(* Visualisation SCHO2_GR4
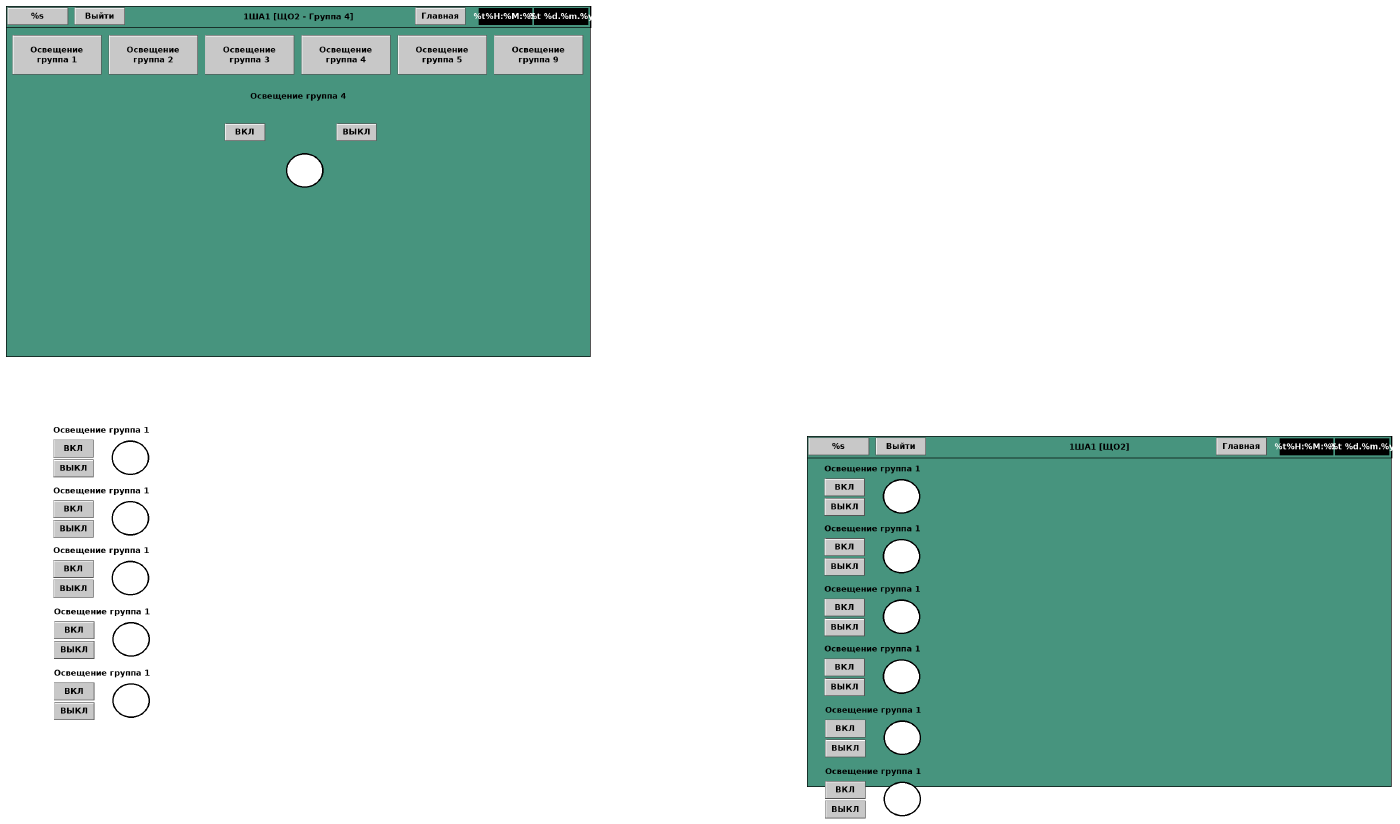
rectangle at (0,0)-(802,30): text "1ША1 [ЩО2 - Группа 4]"
button at (2,2)-(85,26): text "%s"; shows VHOD.User
button at (94,2)-(163,26): text "Выйти"; toggles VHOD.bVihod; opens A0_START_WINDOW
button at (561,2)-(630,26): text "Главная"; opens A1_START_WINDOW
rectangle at (648,3)-(721,26): text "%t%H:%M:%S"
rectangle at (724,3)-(798,26): text "%t %d.%m.%y"
rectangle at (6,107)-(796,141): text "Освещение группа 4"
button at (300,161)-(355,185): text "ВКЛ"; toggles .bK152_1SHA1_SCHO2_LIGHT_GR4_ON
button at (453,161)-(508,185): text "ВЫКЛ"; taps .bK152_1SHA1_SCHO2_LIGHT_GR4_OFF
ellipse at (384,202)-(435,249): alarm colour if .K152_1SHA1_SCHO2_KM_GR4
rectangle at (45,570)-(217,594): text "Освещение группа 1"
button at (65,595)-(120,619): text "ВКЛ"; toggles .bK152_1SHA1_SCHAO1_LIGHT_GR5_ON
button at (65,622)-(120,646): text "ВЫКЛ"; taps .bK152_1SHA1_SCHAO1_LIGHT_GR5_OFF
ellipse at (145,596)-(196,643): alarm colour if .K152_1SHA1_SCHAO1_LIGHT_GR5
rectangle at (45,653)-(217,677): text "Освещение группа 1"
button at (65,678)-(120,702): text "ВКЛ"; toggles .bK152_1SHA1_SCHAO1_LIGHT_GR5_ON
button at (65,705)-(120,729): text "ВЫКЛ"; taps .bK152_1SHA1_SCHAO1_LIGHT_GR5_OFF
ellipse at (145,679)-(196,726): alarm colour if .K152_1SHA1_SCHAO1_LIGHT_GR5
rectangle at (45,735)-(217,759): text "Освещение группа 1"
button at (65,760)-(120,784): text "ВКЛ"; toggles .bK152_1SHA1_SCHAO1_LIGHT_GR5_ON
button at (65,787)-(120,811): text "ВЫКЛ"; taps .bK152_1SHA1_SCHAO1_LIGHT_GR5_OFF
ellipse at (145,761)-(196,808): alarm colour if .K152_1SHA1_SCHAO1_LIGHT_GR5
rectangle at (46,819)-(218,843): text "Освещение группа 1"
button at (66,844)-(121,868): text "ВКЛ"; toggles .bK152_1SHA1_SCHAO1_LIGHT_GR5_ON
button at (66,871)-(121,895): text "ВЫКЛ"; taps .bK152_1SHA1_SCHAO1_LIGHT_GR5_OFF
ellipse at (146,845)-(197,892): alarm colour if .K152_1SHA1_SCHAO1_LIGHT_GR5
rectangle at (46,903)-(218,927): text "Освещение группа 1"
button at (66,928)-(121,952): text "ВКЛ"; toggles .bK152_1SHA1_SCHAO1_LIGHT_GR5_ON
button at (66,955)-(121,979): text "ВЫКЛ"; taps .bK152_1SHA1_SCHAO1_LIGHT_GR5_OFF
ellipse at (146,929)-(197,976): alarm colour if .K152_1SHA1_SCHAO1_LIGHT_GR5
rectangle at (1098,590)-(1900,620): text "1ША1 [ЩО2]"
button at (1100,592)-(1183,616): text "%s"; shows VHOD.User
button at (1192,592)-(1261,616): text "Выйти"; toggles VHOD.bVihod; opens A0_START_WINDOW
button at (1659,592)-(1728,616): text "Главная"; opens A1_START_WINDOW
rectangle at (1746,593)-(1819,616): text "%t%H:%M:%S"
rectangle at (1822,593)-(1896,616): text "%t %d.%m.%y"
rectangle at (1102,623)-(1274,647): text "Освещение группа 1"
button at (1122,648)-(1177,672): text "ВКЛ"; toggles .bK152_1SHA1_SCHAO1_LIGHT_GR5_ON
button at (1122,675)-(1177,699): text "ВЫКЛ"; taps .bK152_1SHA1_SCHAO1_LIGHT_GR5_OFF
ellipse at (1202,649)-(1253,696): alarm colour if .K152_1SHA1_SCHAO1_LIGHT_GR5
rectangle at (1102,705)-(1274,729): text "Освещение группа 1"
button at (1122,730)-(1177,754): text "ВКЛ"; toggles .bK152_1SHA1_SCHAO1_LIGHT_GR5_ON
button at (1122,757)-(1177,781): text "ВЫКЛ"; taps .bK152_1SHA1_SCHAO1_LIGHT_GR5_OFF
ellipse at (1202,731)-(1253,778): alarm colour if .K152_1SHA1_SCHAO1_LIGHT_GR5
rectangle at (1102,788)-(1274,812): text "Освещение группа 1"
button at (1122,813)-(1177,837): text "ВКЛ"; toggles .bK152_1SHA1_SCHAO1_LIGHT_GR5_ON
button at (1122,840)-(1177,864): text "ВЫКЛ"; taps .bK152_1SHA1_SCHAO1_LIGHT_GR5_OFF
ellipse at (1202,814)-(1253,861): alarm colour if .K152_1SHA1_SCHAO1_LIGHT_GR5
rectangle at (1102,870)-(1274,894): text "Освещение группа 1"
button at (1122,895)-(1177,919): text "ВКЛ"; toggles .bK152_1SHA1_SCHAO1_LIGHT_GR5_ON
button at (1122,922)-(1177,946): text "ВЫКЛ"; taps .bK152_1SHA1_SCHAO1_LIGHT_GR5_OFF
ellipse at (1202,896)-(1253,943): alarm colour if .K152_1SHA1_SCHAO1_LIGHT_GR5
rectangle at (1103,954)-(1275,978): text "Освещение группа 1"
button at (1123,979)-(1178,1003): text "ВКЛ"; toggles .bK152_1SHA1_SCHAO1_LIGHT_GR5_ON
button at (1123,1006)-(1178,1030): text "ВЫКЛ"; taps .bK152_1SHA1_SCHAO1_LIGHT_GR5_OFF
ellipse at (1203,980)-(1254,1027): alarm colour if .K152_1SHA1_SCHAO1_LIGHT_GR5
rectangle at (1103,1038)-(1275,1062): text "Освещение группа 1"
button at (1123,1063)-(1178,1087): text "ВКЛ"; toggles .bK152_1SHA1_SCHAO1_LIGHT_GR5_ON
button at (1123,1090)-(1178,1114): text "ВЫКЛ"; taps .bK152_1SHA1_SCHAO1_LIGHT_GR5_OFF
ellipse at (1203,1064)-(1254,1111): alarm colour if .K152_1SHA1_SCHAO1_LIGHT_GR5
button at (9,40)-(131,94): text "Освещение / группа 1"; opens SCHO2_GR1
button at (141,40)-(263,94): text "Освещение / группа 2"; opens SCHO2_GR2
button at (273,40)-(395,94): text "Освещение / группа 3"; opens SCHO2_GR3
button at (405,40)-(527,94): text "Освещение / группа 4"; opens SCHO2_GR4
button at (537,40)-(659,94): text "Освещение / группа 5"; opens SCHO2_GR5
button at (669,40)-(791,94): text "Освещение / группа 9"; opens SCHO2_GR9
2 more shapes without text or variables
14 elements of other kinds (tables, trends, ...) not read
*)

(* Visualisation SCHO2_GR5
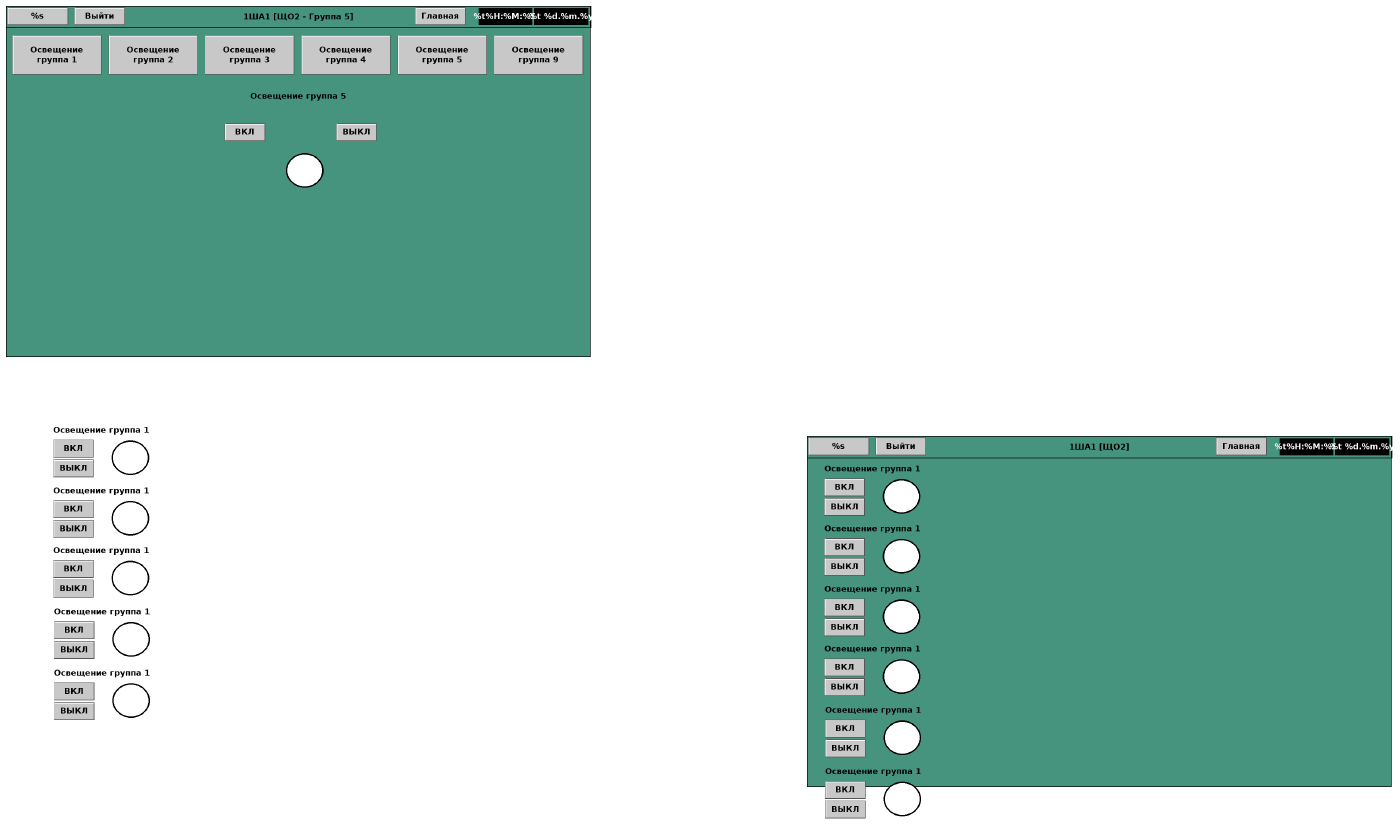
rectangle at (0,0)-(802,30): text "1ША1 [ЩО2 - Группа 5]"
button at (2,2)-(85,26): text "%s"; shows VHOD.User
button at (94,2)-(163,26): text "Выйти"; toggles VHOD.bVihod; opens A0_START_WINDOW
button at (561,2)-(630,26): text "Главная"; opens A1_START_WINDOW
rectangle at (648,3)-(721,26): text "%t%H:%M:%S"
rectangle at (724,3)-(798,26): text "%t %d.%m.%y"
rectangle at (6,107)-(796,141): text "Освещение группа 5"
button at (300,161)-(355,185): text "ВКЛ"; toggles .bK152_1SHA1_SCHO2_LIGHT_GR5_ON
button at (453,161)-(508,185): text "ВЫКЛ"; taps .bK152_1SHA1_SCHO2_LIGHT_GR5_OFF
ellipse at (384,202)-(435,249): alarm colour if .K152_1SHA1_SCHO2_KM_GR5
rectangle at (45,570)-(217,594): text "Освещение группа 1"
button at (65,595)-(120,619): text "ВКЛ"; toggles .bK152_1SHA1_SCHAO1_LIGHT_GR5_ON
button at (65,622)-(120,646): text "ВЫКЛ"; taps .bK152_1SHA1_SCHAO1_LIGHT_GR5_OFF
ellipse at (145,596)-(196,643): alarm colour if .K152_1SHA1_SCHAO1_LIGHT_GR5
rectangle at (45,653)-(217,677): text "Освещение группа 1"
button at (65,678)-(120,702): text "ВКЛ"; toggles .bK152_1SHA1_SCHAO1_LIGHT_GR5_ON
button at (65,705)-(120,729): text "ВЫКЛ"; taps .bK152_1SHA1_SCHAO1_LIGHT_GR5_OFF
ellipse at (145,679)-(196,726): alarm colour if .K152_1SHA1_SCHAO1_LIGHT_GR5
rectangle at (45,735)-(217,759): text "Освещение группа 1"
button at (65,760)-(120,784): text "ВКЛ"; toggles .bK152_1SHA1_SCHAO1_LIGHT_GR5_ON
button at (65,787)-(120,811): text "ВЫКЛ"; taps .bK152_1SHA1_SCHAO1_LIGHT_GR5_OFF
ellipse at (145,761)-(196,808): alarm colour if .K152_1SHA1_SCHAO1_LIGHT_GR5
rectangle at (46,819)-(218,843): text "Освещение группа 1"
button at (66,844)-(121,868): text "ВКЛ"; toggles .bK152_1SHA1_SCHAO1_LIGHT_GR5_ON
button at (66,871)-(121,895): text "ВЫКЛ"; taps .bK152_1SHA1_SCHAO1_LIGHT_GR5_OFF
ellipse at (146,845)-(197,892): alarm colour if .K152_1SHA1_SCHAO1_LIGHT_GR5
rectangle at (46,903)-(218,927): text "Освещение группа 1"
button at (66,928)-(121,952): text "ВКЛ"; toggles .bK152_1SHA1_SCHAO1_LIGHT_GR5_ON
button at (66,955)-(121,979): text "ВЫКЛ"; taps .bK152_1SHA1_SCHAO1_LIGHT_GR5_OFF
ellipse at (146,929)-(197,976): alarm colour if .K152_1SHA1_SCHAO1_LIGHT_GR5
rectangle at (1098,590)-(1900,620): text "1ША1 [ЩО2]"
button at (1100,592)-(1183,616): text "%s"; shows VHOD.User
button at (1192,592)-(1261,616): text "Выйти"; toggles VHOD.bVihod; opens A0_START_WINDOW
button at (1659,592)-(1728,616): text "Главная"; opens A1_START_WINDOW
rectangle at (1746,593)-(1819,616): text "%t%H:%M:%S"
rectangle at (1822,593)-(1896,616): text "%t %d.%m.%y"
rectangle at (1102,623)-(1274,647): text "Освещение группа 1"
button at (1122,648)-(1177,672): text "ВКЛ"; toggles .bK152_1SHA1_SCHAO1_LIGHT_GR5_ON
button at (1122,675)-(1177,699): text "ВЫКЛ"; taps .bK152_1SHA1_SCHAO1_LIGHT_GR5_OFF
ellipse at (1202,649)-(1253,696): alarm colour if .K152_1SHA1_SCHAO1_LIGHT_GR5
rectangle at (1102,705)-(1274,729): text "Освещение группа 1"
button at (1122,730)-(1177,754): text "ВКЛ"; toggles .bK152_1SHA1_SCHAO1_LIGHT_GR5_ON
button at (1122,757)-(1177,781): text "ВЫКЛ"; taps .bK152_1SHA1_SCHAO1_LIGHT_GR5_OFF
ellipse at (1202,731)-(1253,778): alarm colour if .K152_1SHA1_SCHAO1_LIGHT_GR5
rectangle at (1102,788)-(1274,812): text "Освещение группа 1"
button at (1122,813)-(1177,837): text "ВКЛ"; toggles .bK152_1SHA1_SCHAO1_LIGHT_GR5_ON
button at (1122,840)-(1177,864): text "ВЫКЛ"; taps .bK152_1SHA1_SCHAO1_LIGHT_GR5_OFF
ellipse at (1202,814)-(1253,861): alarm colour if .K152_1SHA1_SCHAO1_LIGHT_GR5
rectangle at (1102,870)-(1274,894): text "Освещение группа 1"
button at (1122,895)-(1177,919): text "ВКЛ"; toggles .bK152_1SHA1_SCHAO1_LIGHT_GR5_ON
button at (1122,922)-(1177,946): text "ВЫКЛ"; taps .bK152_1SHA1_SCHAO1_LIGHT_GR5_OFF
ellipse at (1202,896)-(1253,943): alarm colour if .K152_1SHA1_SCHAO1_LIGHT_GR5
rectangle at (1103,954)-(1275,978): text "Освещение группа 1"
button at (1123,979)-(1178,1003): text "ВКЛ"; toggles .bK152_1SHA1_SCHAO1_LIGHT_GR5_ON
button at (1123,1006)-(1178,1030): text "ВЫКЛ"; taps .bK152_1SHA1_SCHAO1_LIGHT_GR5_OFF
ellipse at (1203,980)-(1254,1027): alarm colour if .K152_1SHA1_SCHAO1_LIGHT_GR5
rectangle at (1103,1038)-(1275,1062): text "Освещение группа 1"
button at (1123,1063)-(1178,1087): text "ВКЛ"; toggles .bK152_1SHA1_SCHAO1_LIGHT_GR5_ON
button at (1123,1090)-(1178,1114): text "ВЫКЛ"; taps .bK152_1SHA1_SCHAO1_LIGHT_GR5_OFF
ellipse at (1203,1064)-(1254,1111): alarm colour if .K152_1SHA1_SCHAO1_LIGHT_GR5
button at (9,40)-(131,94): text "Освещение / группа 1"; opens SCHO2_GR1
button at (141,40)-(263,94): text "Освещение / группа 2"; opens SCHO2_GR2
button at (273,40)-(395,94): text "Освещение / группа 3"; opens SCHO2_GR3
button at (405,40)-(527,94): text "Освещение / группа 4"; opens SCHO2_GR4
button at (537,40)-(659,94): text "Освещение / группа 5"; opens SCHO2_GR5
button at (669,40)-(791,94): text "Освещение / группа 9"; opens SCHO2_GR9
2 more shapes without text or variables
14 elements of other kinds (tables, trends, ...) not read
*)

(* Visualisation SCHO2_GR9
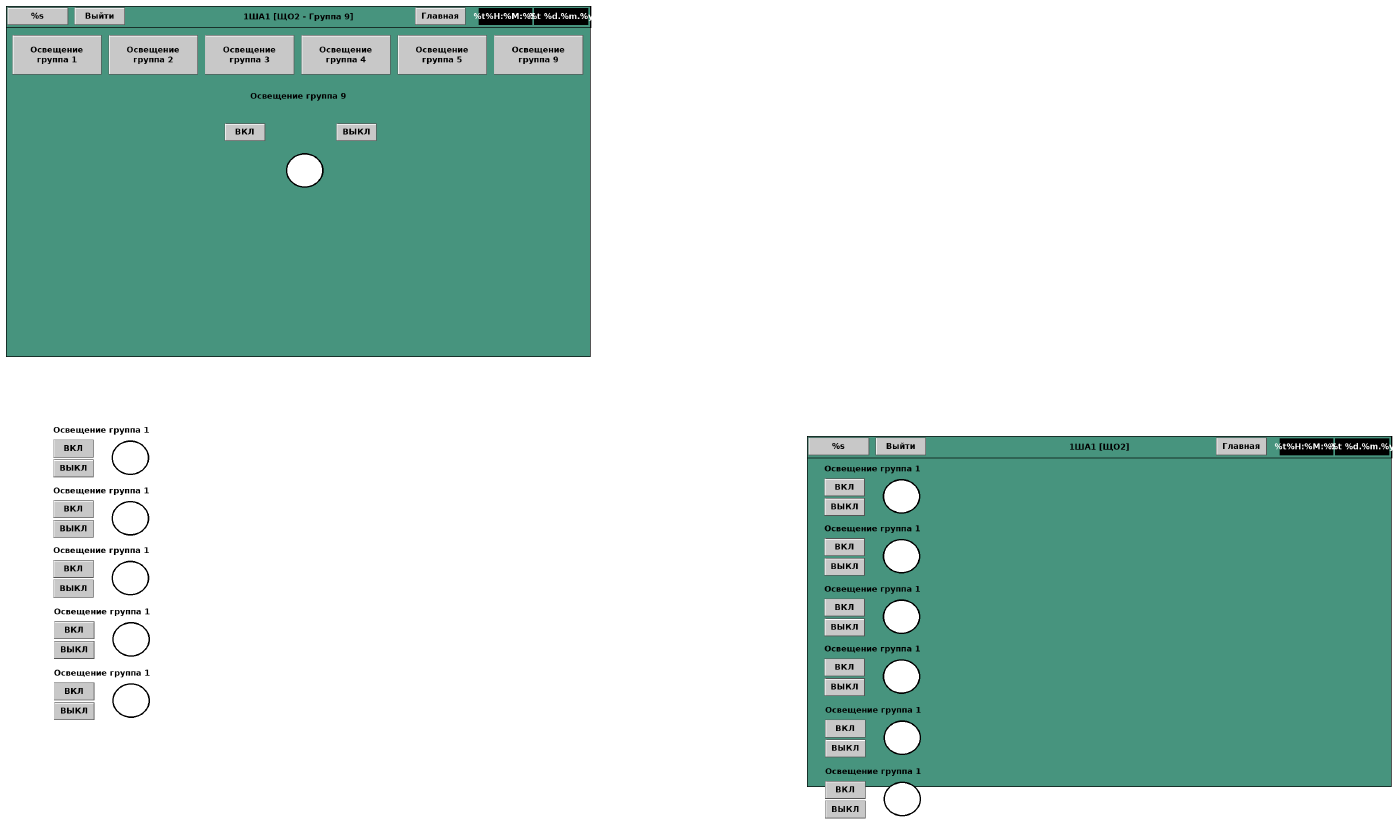
rectangle at (0,0)-(802,30): text "1ША1 [ЩО2 - Группа 9]"
button at (2,2)-(85,26): text "%s"; shows VHOD.User
button at (94,2)-(163,26): text "Выйти"; toggles VHOD.bVihod; opens A0_START_WINDOW
button at (561,2)-(630,26): text "Главная"; opens A1_START_WINDOW
rectangle at (648,3)-(721,26): text "%t%H:%M:%S"
rectangle at (724,3)-(798,26): text "%t %d.%m.%y"
rectangle at (6,107)-(796,141): text "Освещение группа 9"
button at (300,161)-(355,185): text "ВКЛ"; toggles .bK152_1SHA1_SCHO2_LIGHT_GR9_ON
button at (453,161)-(508,185): text "ВЫКЛ"; taps .bK152_1SHA1_SCHO2_LIGHT_GR9_OFF
ellipse at (384,202)-(435,249): alarm colour if .K152_1SHA1_SCHO2_KM_GR9
rectangle at (45,570)-(217,594): text "Освещение группа 1"
button at (65,595)-(120,619): text "ВКЛ"; toggles .bK152_1SHA1_SCHAO1_LIGHT_GR5_ON
button at (65,622)-(120,646): text "ВЫКЛ"; taps .bK152_1SHA1_SCHAO1_LIGHT_GR5_OFF
ellipse at (145,596)-(196,643): alarm colour if .K152_1SHA1_SCHAO1_LIGHT_GR5
rectangle at (45,653)-(217,677): text "Освещение группа 1"
button at (65,678)-(120,702): text "ВКЛ"; toggles .bK152_1SHA1_SCHAO1_LIGHT_GR5_ON
button at (65,705)-(120,729): text "ВЫКЛ"; taps .bK152_1SHA1_SCHAO1_LIGHT_GR5_OFF
ellipse at (145,679)-(196,726): alarm colour if .K152_1SHA1_SCHAO1_LIGHT_GR5
rectangle at (45,735)-(217,759): text "Освещение группа 1"
button at (65,760)-(120,784): text "ВКЛ"; toggles .bK152_1SHA1_SCHAO1_LIGHT_GR5_ON
button at (65,787)-(120,811): text "ВЫКЛ"; taps .bK152_1SHA1_SCHAO1_LIGHT_GR5_OFF
ellipse at (145,761)-(196,808): alarm colour if .K152_1SHA1_SCHAO1_LIGHT_GR5
rectangle at (46,819)-(218,843): text "Освещение группа 1"
button at (66,844)-(121,868): text "ВКЛ"; toggles .bK152_1SHA1_SCHAO1_LIGHT_GR5_ON
button at (66,871)-(121,895): text "ВЫКЛ"; taps .bK152_1SHA1_SCHAO1_LIGHT_GR5_OFF
ellipse at (146,845)-(197,892): alarm colour if .K152_1SHA1_SCHAO1_LIGHT_GR5
rectangle at (46,903)-(218,927): text "Освещение группа 1"
button at (66,928)-(121,952): text "ВКЛ"; toggles .bK152_1SHA1_SCHAO1_LIGHT_GR5_ON
button at (66,955)-(121,979): text "ВЫКЛ"; taps .bK152_1SHA1_SCHAO1_LIGHT_GR5_OFF
ellipse at (146,929)-(197,976): alarm colour if .K152_1SHA1_SCHAO1_LIGHT_GR5
rectangle at (1098,590)-(1900,620): text "1ША1 [ЩО2]"
button at (1100,592)-(1183,616): text "%s"; shows VHOD.User
button at (1192,592)-(1261,616): text "Выйти"; toggles VHOD.bVihod; opens A0_START_WINDOW
button at (1659,592)-(1728,616): text "Главная"; opens A1_START_WINDOW
rectangle at (1746,593)-(1819,616): text "%t%H:%M:%S"
rectangle at (1822,593)-(1896,616): text "%t %d.%m.%y"
rectangle at (1102,623)-(1274,647): text "Освещение группа 1"
button at (1122,648)-(1177,672): text "ВКЛ"; toggles .bK152_1SHA1_SCHAO1_LIGHT_GR5_ON
button at (1122,675)-(1177,699): text "ВЫКЛ"; taps .bK152_1SHA1_SCHAO1_LIGHT_GR5_OFF
ellipse at (1202,649)-(1253,696): alarm colour if .K152_1SHA1_SCHAO1_LIGHT_GR5
rectangle at (1102,705)-(1274,729): text "Освещение группа 1"
button at (1122,730)-(1177,754): text "ВКЛ"; toggles .bK152_1SHA1_SCHAO1_LIGHT_GR5_ON
button at (1122,757)-(1177,781): text "ВЫКЛ"; taps .bK152_1SHA1_SCHAO1_LIGHT_GR5_OFF
ellipse at (1202,731)-(1253,778): alarm colour if .K152_1SHA1_SCHAO1_LIGHT_GR5
rectangle at (1102,788)-(1274,812): text "Освещение группа 1"
button at (1122,813)-(1177,837): text "ВКЛ"; toggles .bK152_1SHA1_SCHAO1_LIGHT_GR5_ON
button at (1122,840)-(1177,864): text "ВЫКЛ"; taps .bK152_1SHA1_SCHAO1_LIGHT_GR5_OFF
ellipse at (1202,814)-(1253,861): alarm colour if .K152_1SHA1_SCHAO1_LIGHT_GR5
rectangle at (1102,870)-(1274,894): text "Освещение группа 1"
button at (1122,895)-(1177,919): text "ВКЛ"; toggles .bK152_1SHA1_SCHAO1_LIGHT_GR5_ON
button at (1122,922)-(1177,946): text "ВЫКЛ"; taps .bK152_1SHA1_SCHAO1_LIGHT_GR5_OFF
ellipse at (1202,896)-(1253,943): alarm colour if .K152_1SHA1_SCHAO1_LIGHT_GR5
rectangle at (1103,954)-(1275,978): text "Освещение группа 1"
button at (1123,979)-(1178,1003): text "ВКЛ"; toggles .bK152_1SHA1_SCHAO1_LIGHT_GR5_ON
button at (1123,1006)-(1178,1030): text "ВЫКЛ"; taps .bK152_1SHA1_SCHAO1_LIGHT_GR5_OFF
ellipse at (1203,980)-(1254,1027): alarm colour if .K152_1SHA1_SCHAO1_LIGHT_GR5
rectangle at (1103,1038)-(1275,1062): text "Освещение группа 1"
button at (1123,1063)-(1178,1087): text "ВКЛ"; toggles .bK152_1SHA1_SCHAO1_LIGHT_GR5_ON
button at (1123,1090)-(1178,1114): text "ВЫКЛ"; taps .bK152_1SHA1_SCHAO1_LIGHT_GR5_OFF
ellipse at (1203,1064)-(1254,1111): alarm colour if .K152_1SHA1_SCHAO1_LIGHT_GR5
button at (9,40)-(131,94): text "Освещение / группа 1"; opens SCHO2_GR1
button at (141,40)-(263,94): text "Освещение / группа 2"; opens SCHO2_GR2
button at (273,40)-(395,94): text "Освещение / группа 3"; opens SCHO2_GR3
button at (405,40)-(527,94): text "Освещение / группа 4"; opens SCHO2_GR4
button at (537,40)-(659,94): text "Освещение / группа 5"; opens SCHO2_GR5
button at (669,40)-(791,94): text "Освещение / группа 9"; opens SCHO2_GR9
2 more shapes without text or variables
14 elements of other kinds (tables, trends, ...) not read
*)

(* Visualisation SYSTEM_CONDITIONING
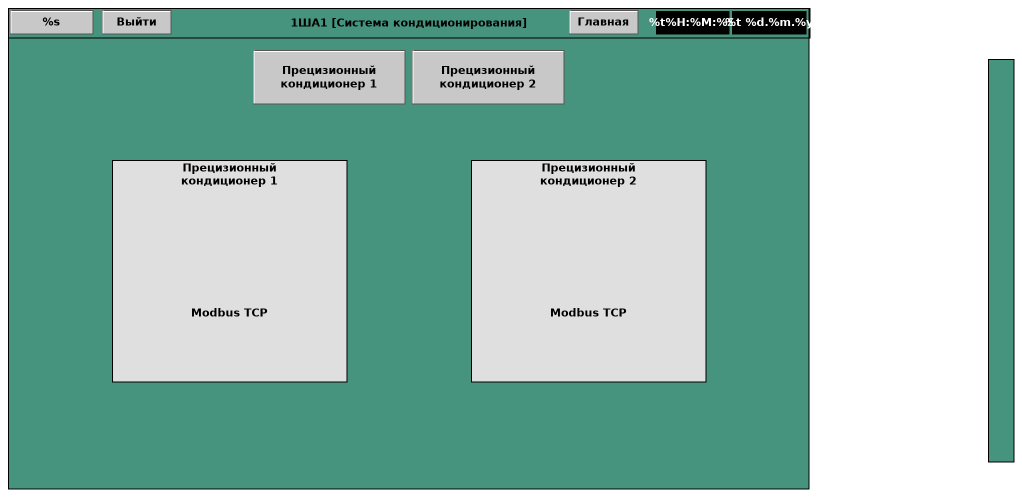
rectangle at (0,0)-(802,30): text "1ША1 [Система кондиционирования]"
button at (2,2)-(85,26): text "%s"; shows VHOD.User
button at (94,2)-(163,26): text "Выйти"; toggles VHOD.bVihod; opens A0_START_WINDOW
button at (561,2)-(630,26): text "Главная"; opens A1_START_WINDOW
rectangle at (648,3)-(721,26): text "%t%H:%M:%S"
rectangle at (724,3)-(798,26): text "%t %d.%m.%y"
button at (245,42)-(397,96): text "Прецизионный / кондиционер 1"
button at (404,42)-(556,96): text "Прецизионный / кондиционер 2"
rectangle at (104,152)-(339,374): text "Прецизионный / кондиционер 1 /  /  /  /  /  /  /  /  /  / Modbus TCP"
rectangle at (463,152)-(698,374): text "Прецизионный / кондиционер 2 /  /  /  /  /  /  /  /  /  / Modbus TCP"
2 more shapes without text or variables
*)

(* Visualisation SYSTEM_GAS_CONTROL
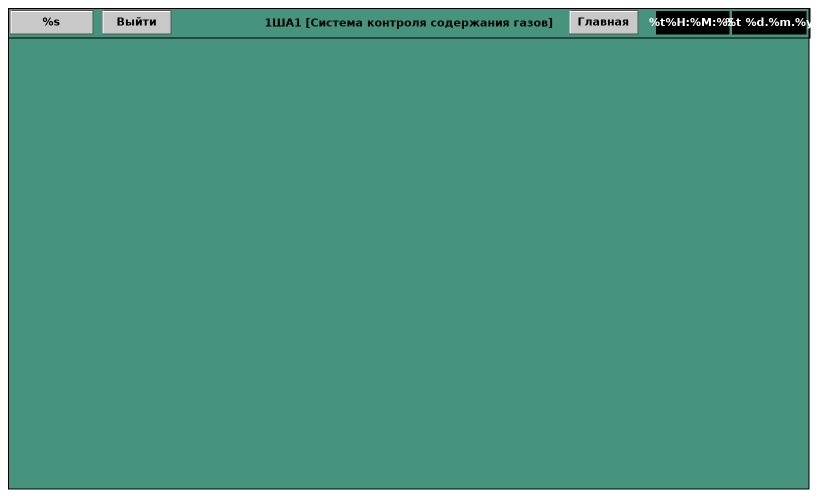
rectangle at (0,0)-(802,30): text "1ША1 [Система контроля содержания газов]"
button at (2,2)-(85,26): text "%s"; shows VHOD.User
button at (94,2)-(163,26): text "Выйти"; toggles VHOD.bVihod; opens A0_START_WINDOW
button at (561,2)-(630,26): text "Главная"; opens A1_START_WINDOW
rectangle at (648,3)-(721,26): text "%t%H:%M:%S"
rectangle at (724,3)-(798,26): text "%t %d.%m.%y"
1 more shapes without text or variables
*)

(* Visualisation SYSTEM_WATER_SUPPLY
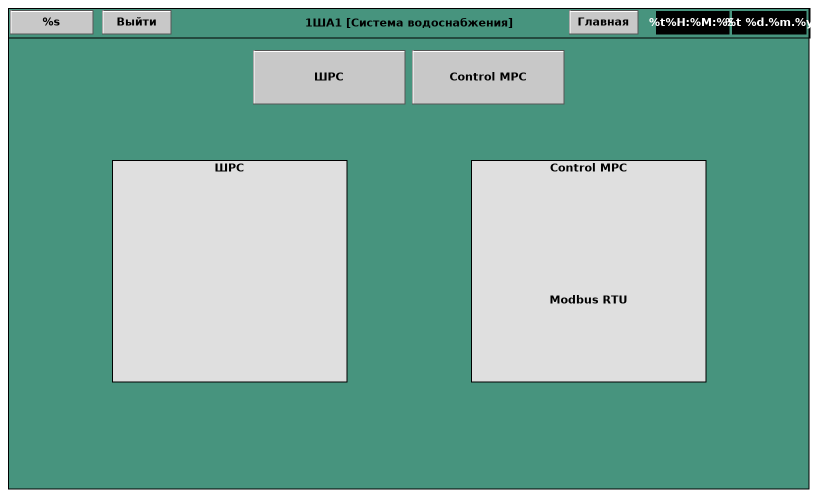
rectangle at (0,0)-(802,30): text "1ША1 [Система водоснабжения]"
button at (2,2)-(85,26): text "%s"; shows VHOD.User
button at (94,2)-(163,26): text "Выйти"; toggles VHOD.bVihod; opens A0_START_WINDOW
button at (561,2)-(630,26): text "Главная"; opens A1_START_WINDOW
rectangle at (648,3)-(721,26): text "%t%H:%M:%S"
rectangle at (724,3)-(798,26): text "%t %d.%m.%y"
button at (245,42)-(397,96): text "ШРС"
button at (404,42)-(556,96): text "Control MPC"
rectangle at (104,152)-(339,374): text "ШРС"
rectangle at (463,152)-(698,374): text "Control MPC /  /  /  /  /  /  /  /  /  / Modbus RTU"
1 more shapes without text or variables
*)

(* Visualisation TEMP_CONTROL
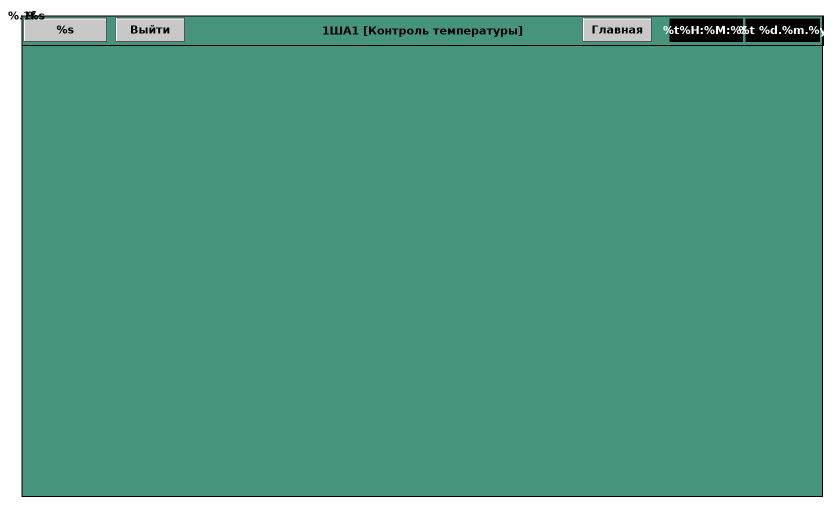
rectangle at (0,0)-(802,30): text "1ША1 [Контроль температуры]"
button at (2,2)-(85,26): text "%s"; shows VHOD.User
button at (94,2)-(163,26): text "Выйти"; toggles VHOD.bVihod; opens A0_START_WINDOW
button at (561,2)-(630,26): text "Главная"; opens A1_START_WINDOW
rectangle at (0,0)-(0,0): text "%s"; shows masTABLE_TEMPERATURE[INDEX].s1Positioin
rectangle at (0,0)-(0,0): text "%.1f"; shows masTABLE_TEMPERATURE[INDEX].s2Value
rectangle at (648,3)-(721,26): text "%t%H:%M:%S"
rectangle at (724,3)-(798,26): text "%t %d.%m.%y"
1 more shapes without text or variables
*)

(* Visualisation test_weekly
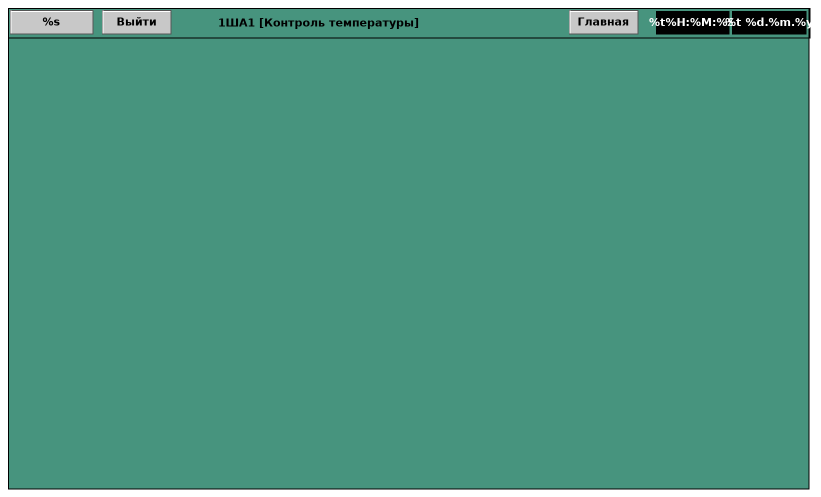
rectangle at (0,0)-(802,30): text "1ША1 [Контроль температуры]"
button at (2,2)-(85,26): text "%s"; shows VHOD.User
button at (94,2)-(163,26): text "Выйти"; toggles VHOD.bVihod; opens A0_START_WINDOW
button at (561,2)-(630,26): text "Главная"; opens A1_START_WINDOW
rectangle at (648,3)-(721,26): text "%t%H:%M:%S"
rectangle at (724,3)-(798,26): text "%t %d.%m.%y"
1 more shapes without text or variables
1 elements of other kinds (tables, trends, ...) not read
*)
